// TIA Portal V18 program export: 2 tag tables, 0 data types, 2 data blocks, 2 code blocks (in call order from the OBs), 0 instance data blocks

VAR_GLOBAL   // PLC tag table "Default tag table"
   Motor_Contactor AT %Q0.0 : Bool;
   Clock_Byte AT %MB100 : Byte;
   Clock_10Hz AT %M100.0 : Bool;
   Clock_5Hz AT %M100.1 : Bool;
   "Clock_2.5Hz" AT %M100.2 : Bool;
   Clock_2Hz AT %M100.3 : Bool;
   "Clock_1.25Hz" AT %M100.4 : Bool;
   "Clock_0.625Hz" AT %M100.6 : Bool;
   "Clock_0.5Hz" AT %M100.7 : Bool;
END_VAR

VAR_GLOBAL   // PLC tag table "PLC2_Tags"
   MB_ControlWord AT %MW40 : Word;
   MB_FreqSetpoint AT %MW42 : Int;
   MB_StatusWord AT %MW44 : Word;
   MB_ActualSpeed AT %MW46 : Int;
   MB_Error AT %M50.0 : Bool;
   MB_Busy AT %M50.1 : Bool;
   MB_Done AT %M50.2 : Bool;
   MB_Status AT %MW52 : Word;
   iStep AT %MW60 : Int;
   Freq_Temp AT %MD70 : Real;
   Speed_Actual_Temp AT %MD74 : Real;
   FirstScan AT %M101.0 : Bool;
   Clock_1Hz AT %M100.5 : Bool;
   MBCL_Done AT %M51.0 : Bool;
   MBCL_Error AT %M51.1 : Bool;
   MBCL_Status AT %MW54 : Word;
END_VAR

DATA_BLOCK "DB1_NhanTuPLC1"   // DB1
{ S7_Optimized_Access := 'FALSE' }
VERSION : 0.1
// stored: AutoNumber true, IsOnlyStoredInLoadMemory false, IsWriteProtectedInAS false
   VAR
      Speed_SP_fromPLC1 : Real;
      Control_Byte : Bool;
      Reset_Cmd : Bool;
      DIR_Cmd : Bool;
   END_VAR
BEGIN
END_DATA_BLOCK

DATA_BLOCK "DB2_GuiVePLC1"   // DB2
{ S7_Optimized_Access := 'FALSE' }
VERSION : 0.1
// stored: AutoNumber true, IsOnlyStoredInLoadMemory false, IsWriteProtectedInAS false
   VAR
      Speed_Actual_toSend : Real;
      ATV12_Status_toSend : Word;
   END_VAR
BEGIN
END_DATA_BLOCK

ORGANIZATION_BLOCK "Main"   // OB1, LAD, ProgramCycle
TITLE = "Main Program Sweep (Cycle)"
{ S7_Optimized_Access := 'TRUE' }
VERSION : 0.1
// stored: AutoNumber true, IsIECCheckEnabled false, SetENOAutomatically false
   VAR_INPUT
      Initial_Call : Bool;   // Initial call of this OB
      Remanence : Bool;   // =True, if remanent data are available
   END_VAR
BEGIN

REGION Network 1: Call FC_PLC2_Logic (Convert + Step Advance)
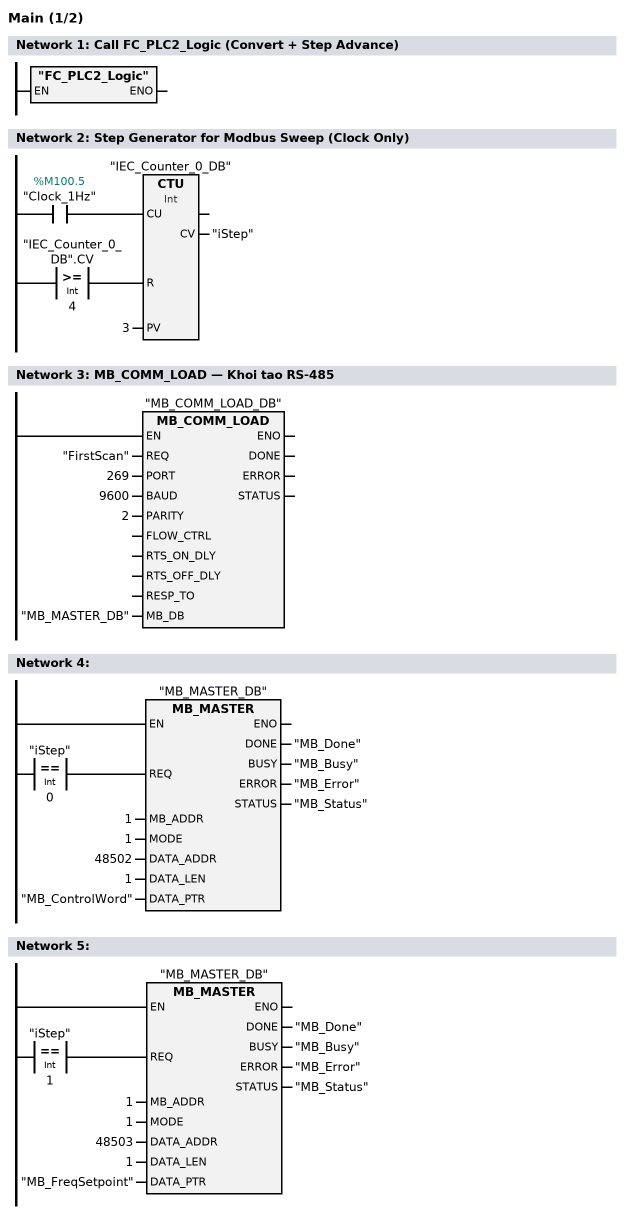
   RUNG wire#powerrail
      "FC_PLC2_Logic"()
   END_RUNG
   // the same network as SCL:
   "FC_PLC2_Logic"();
END_REGION

REGION Network 2: Step Generator for Modbus Sweep (Clock Only)
   RUNG wire#powerrail
      Contact( "Clock_1Hz" )
      { S7_Templates := "value_type := Int" } "IEC_Counter_0_DB".CTU(r := wire#w1, pv := 3, cv => "iStep")
   END_RUNG
   RUNG wire#powerrail
      { S7_Templates := "SrcType := Int" } GE_Contact(in1 := "IEC_Counter_0_DB".CV, in2 := 4)
   END_RUNG wire#w1
   // the same network as SCL:
   "IEC_Counter_0_DB".CTU(CU := "Clock_1Hz", R := "IEC_Counter_0_DB".CV >= 4, PV := 3, CV => "iStep");
END_REGION

REGION Network 3: MB_COMM_LOAD — Khoi tao RS-485
   RUNG wire#powerrail
      "MB_COMM_LOAD_DB".MB_COMM_LOAD(REQ := "FirstScan", PORT := 269, BAUD := 9600, PARITY := 2, FLOW_CTRL :=, RTS_ON_DLY :=, RTS_OFF_DLY :=, RESP_TO :=, MB_DB := "MB_MASTER_DB", DONE =>, ERROR =>, STATUS =>)
   END_RUNG
   // the same network as SCL:
   "MB_COMM_LOAD_DB"(REQ := "FirstScan", PORT := 269, BAUD := 9600, PARITY := 2, MB_DB := "MB_MASTER_DB");   // MB_COMM_LOAD
END_REGION

REGION Network 4
   RUNG wire#powerrail
      "MB_MASTER_DB".MB_MASTER(REQ := wire#w1, MB_ADDR := 1, MODE := 1, DATA_ADDR := 48502, DATA_LEN := 1, DATA_PTR := "MB_ControlWord", DONE => "MB_Done", BUSY => "MB_Busy", ERROR => "MB_Error", STATUS => "MB_Status")
   END_RUNG
   RUNG wire#powerrail
      { S7_Templates := "SrcType := Int" } EQ_Contact(in1 := "iStep", in2 := 0)
   END_RUNG wire#w1
   // the same network as SCL:
   "MB_MASTER_DB"(REQ := "iStep" = 0,   // MB_MASTER
                  MB_ADDR := 1,
                  MODE := 1,
                  DATA_ADDR := 48502,
                  DATA_LEN := 1,
                  DATA_PTR := "MB_ControlWord",
                  DONE => "MB_Done",
                  BUSY => "MB_Busy",
                  ERROR => "MB_Error",
                  STATUS => "MB_Status");
END_REGION

REGION Network 5
   RUNG wire#powerrail
      "MB_MASTER_DB".MB_MASTER(REQ := wire#w1, MB_ADDR := 1, MODE := 1, DATA_ADDR := 48503, DATA_LEN := 1, DATA_PTR := "MB_FreqSetpoint", DONE => "MB_Done", BUSY => "MB_Busy", ERROR => "MB_Error", STATUS => "MB_Status")
   END_RUNG
   RUNG wire#powerrail
      { S7_Templates := "SrcType := Int" } EQ_Contact(in1 := "iStep", in2 := 1)
   END_RUNG wire#w1
   // the same network as SCL:
   "MB_MASTER_DB"(REQ := "iStep" = 1,   // MB_MASTER
                  MB_ADDR := 1,
                  MODE := 1,
                  DATA_ADDR := 48503,
                  DATA_LEN := 1,
                  DATA_PTR := "MB_FreqSetpoint",
                  DONE => "MB_Done",
                  BUSY => "MB_Busy",
                  ERROR => "MB_Error",
                  STATUS => "MB_Status");
END_REGION

REGION Network 6
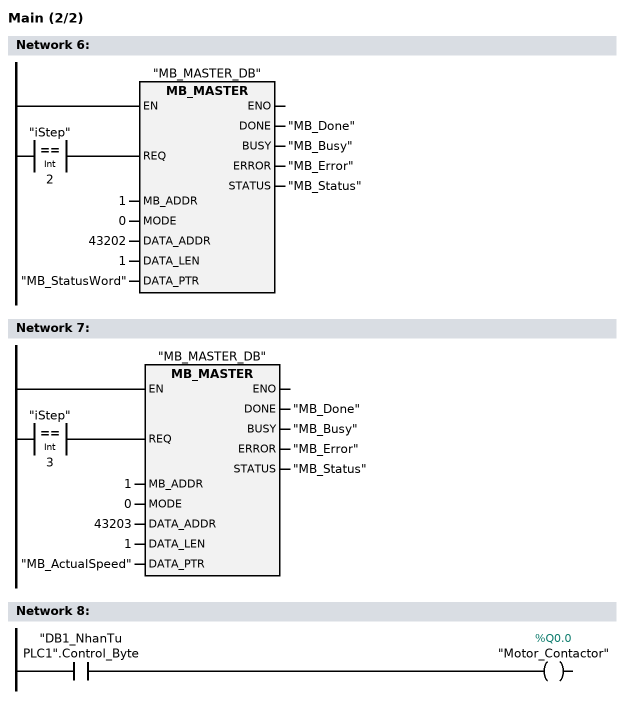
   RUNG wire#powerrail
      "MB_MASTER_DB".MB_MASTER(REQ := wire#w1, MB_ADDR := 1, MODE := 0, DATA_ADDR := 43202, DATA_LEN := 1, DATA_PTR := "MB_StatusWord", DONE => "MB_Done", BUSY => "MB_Busy", ERROR => "MB_Error", STATUS => "MB_Status")
   END_RUNG
   RUNG wire#powerrail
      { S7_Templates := "SrcType := Int" } EQ_Contact(in1 := "iStep", in2 := 2)
   END_RUNG wire#w1
   // the same network as SCL:
   "MB_MASTER_DB"(REQ := "iStep" = 2,   // MB_MASTER
                  MB_ADDR := 1,
                  MODE := 0,
                  DATA_ADDR := 43202,
                  DATA_LEN := 1,
                  DATA_PTR := "MB_StatusWord",
                  DONE => "MB_Done",
                  BUSY => "MB_Busy",
                  ERROR => "MB_Error",
                  STATUS => "MB_Status");
END_REGION

REGION Network 7
   RUNG wire#powerrail
      "MB_MASTER_DB".MB_MASTER(REQ := wire#w1, MB_ADDR := 1, MODE := 0, DATA_ADDR := 43203, DATA_LEN := 1, DATA_PTR := "MB_ActualSpeed", DONE => "MB_Done", BUSY => "MB_Busy", ERROR => "MB_Error", STATUS => "MB_Status")
   END_RUNG
   RUNG wire#powerrail
      { S7_Templates := "SrcType := Int" } EQ_Contact(in1 := "iStep", in2 := 3)
   END_RUNG wire#w1
   // the same network as SCL:
   "MB_MASTER_DB"(REQ := "iStep" = 3,   // MB_MASTER
                  MB_ADDR := 1,
                  MODE := 0,
                  DATA_ADDR := 43203,
                  DATA_LEN := 1,
                  DATA_PTR := "MB_ActualSpeed",
                  DONE => "MB_Done",
                  BUSY => "MB_Busy",
                  ERROR => "MB_Error",
                  STATUS => "MB_Status");
END_REGION

REGION Network 8
   RUNG wire#powerrail
      Contact( "DB1_NhanTuPLC1".Control_Byte )
      Coil( "Motor_Contactor" )
   END_RUNG
   // the same network as SCL:
   "Motor_Contactor" := "DB1_NhanTuPLC1".Control_Byte;
END_REGION
END_ORGANIZATION_BLOCK

FUNCTION "FC_PLC2_Logic" : Void   // FC10, LAD
{ S7_Optimized_Access := 'TRUE' }
VERSION : 0.1
// stored: AutoNumber true, IsIECCheckEnabled false, SetENOAutomatically false, UDAEnableTagReadback false
BEGIN

REGION Network 1: Freq Scale: SP x 10
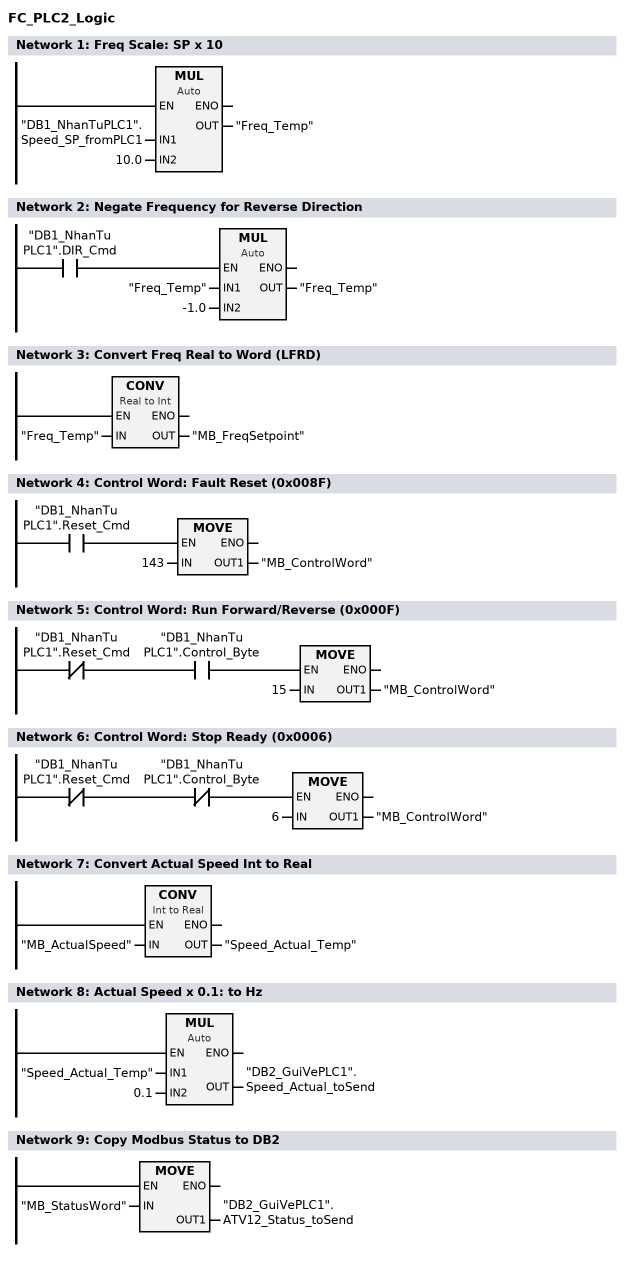
   RUNG wire#powerrail
      { S7_GenerateENO := "TRUE" } Mul(in1 := "DB1_NhanTuPLC1".Speed_SP_fromPLC1, in2 := 10.0, out => "Freq_Temp")
   END_RUNG
   // the same network as SCL:
   "Freq_Temp" := "DB1_NhanTuPLC1".Speed_SP_fromPLC1 * 10.0;
END_REGION

REGION Network 2: Negate Frequency for Reverse Direction
   RUNG wire#powerrail
      Contact( "DB1_NhanTuPLC1".DIR_Cmd )
      { S7_GenerateENO := "TRUE" } Mul(in1 := "Freq_Temp", in2 := -1.0, out => "Freq_Temp")
   END_RUNG
   // the same network as SCL:
   IF "DB1_NhanTuPLC1".DIR_Cmd THEN "Freq_Temp" := "Freq_Temp" * (-1.0); END_IF;
END_REGION

REGION Network 3: Convert Freq Real to Word (LFRD)
   RUNG wire#powerrail
      { S7_Templates := "[SrcType := Real, DestType := Int]"; S7_GenerateENO := "TRUE" } Convert(in := "Freq_Temp", out => "MB_FreqSetpoint")
   END_RUNG
   // the same network as SCL:
   "MB_FreqSetpoint" := REAL_TO_INT("Freq_Temp");
END_REGION

REGION Network 4: Control Word: Fault Reset (0x008F)
   RUNG wire#powerrail
      Contact( "DB1_NhanTuPLC1".Reset_Cmd )
      { S7_GenerateENO := "TRUE" } Move(in := 143, out1 => "MB_ControlWord")
   END_RUNG
   // the same network as SCL:
   IF "DB1_NhanTuPLC1".Reset_Cmd THEN "MB_ControlWord" := 143; END_IF;
END_REGION

REGION Network 5: Control Word: Run Forward/Reverse (0x000F)
   RUNG wire#powerrail
      I_Contact( "DB1_NhanTuPLC1".Reset_Cmd )
      Contact( "DB1_NhanTuPLC1".Control_Byte )
      { S7_GenerateENO := "TRUE" } Move(in := 15, out1 => "MB_ControlWord")
   END_RUNG
   // the same network as SCL:
   IF NOT "DB1_NhanTuPLC1".Reset_Cmd AND "DB1_NhanTuPLC1".Control_Byte THEN "MB_ControlWord" := 15; END_IF;
END_REGION

REGION Network 6: Control Word: Stop Ready (0x0006)
   RUNG wire#powerrail
      I_Contact( "DB1_NhanTuPLC1".Reset_Cmd )
      I_Contact( "DB1_NhanTuPLC1".Control_Byte )
      { S7_GenerateENO := "TRUE" } Move(in := 6, out1 => "MB_ControlWord")
   END_RUNG
   // the same network as SCL:
   IF NOT "DB1_NhanTuPLC1".Reset_Cmd AND NOT "DB1_NhanTuPLC1".Control_Byte THEN
       "MB_ControlWord" := 6;
   END_IF;
END_REGION

REGION Network 7: Convert Actual Speed Int to Real
   RUNG wire#powerrail
      { S7_Templates := "[SrcType := Int, DestType := Real]"; S7_GenerateENO := "TRUE" } Convert(in := "MB_ActualSpeed", out => "Speed_Actual_Temp")
   END_RUNG
   // the same network as SCL:
   "Speed_Actual_Temp" := INT_TO_REAL("MB_ActualSpeed");
END_REGION

REGION Network 8: Actual Speed x 0.1: to Hz
   RUNG wire#powerrail
      { S7_GenerateENO := "TRUE" } Mul(in1 := "Speed_Actual_Temp", in2 := 0.1, out => "DB2_GuiVePLC1".Speed_Actual_toSend)
   END_RUNG
   // the same network as SCL:
   "DB2_GuiVePLC1".Speed_Actual_toSend := "Speed_Actual_Temp" * 0.1;
END_REGION

REGION Network 9: Copy Modbus Status to DB2
   RUNG wire#powerrail
      { S7_GenerateENO := "TRUE" } Move(in := "MB_StatusWord", out1 => "DB2_GuiVePLC1".ATV12_Status_toSend)
   END_RUNG
   // the same network as SCL:
   "DB2_GuiVePLC1".ATV12_Status_toSend := "MB_StatusWord";
END_REGION
END_FUNCTION
